FUNCTION ReadModbusReal : REAL
VAR
	i: INT;
	modbusReal: ModbusUnion;
END_VAR


i:= GVL.nOutputRegisterIndex;

modbusReal.wordValue[1]:= GVL.mb_Output_Registers[i+0];
modbusReal.wordValue[2]:= GVL.mb_Output_Registers[i+1];

GVL.nOutputRegisterIndex:= i + 2;

ReadModbusReal:=modbusReal.realValue;

END_FUNCTION

(* stored: Version 1.1.0.1, ProductVersion 3.1.4024.12
   POU ReadModbusReal: Id {7a0c48b0-0cf1-456c-a39d-c4b05fddbe23}, SpecialFunc None *)
